ABB RobotStudio station: UiS_E458_nov18_20210914-220803.rsstn

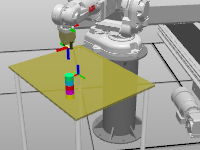
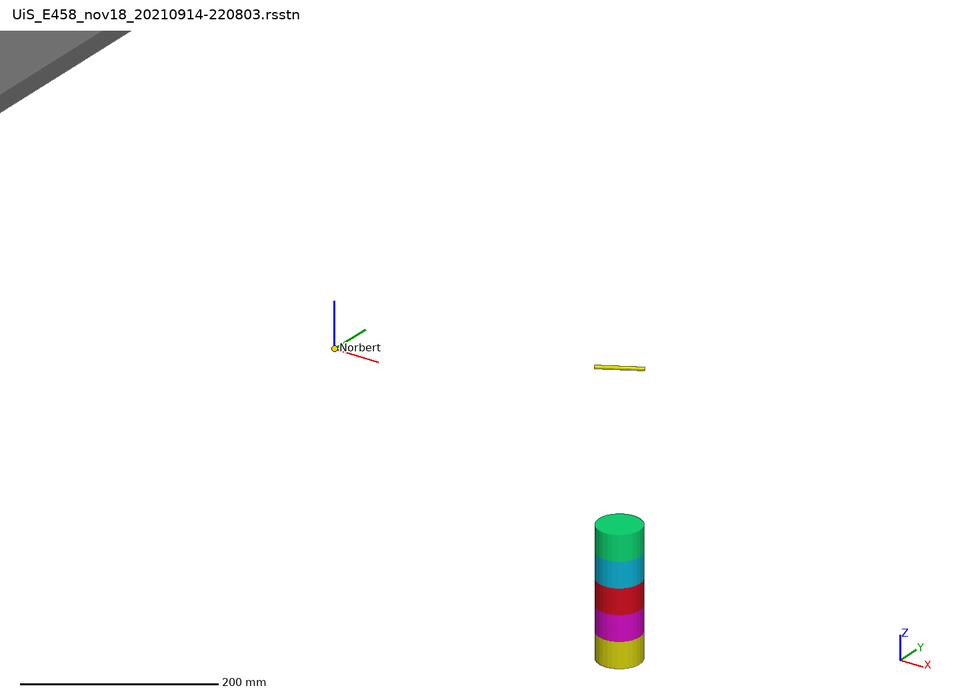
[picture v1: parts stored in the station drawn from their meshes, with robot base, taught points and paths (robot models come from the ABB library and are not in the file)]
Station UiS_E458_nov18 (saved by RobotStudio 21.2.9526.0)
Controller Norbert, task T_ROB1: task frame (RAPID world) sits at (-305, -752, 720) mm, rotated rx 0 ry 0 rz 30 deg in the station
Controller Norbert
  mechanical unit ROB_1: Norbert, 6 joints, base frame (0, 0, 0) mm
Layout (positions relative to the parent item):
  - PedestalN [part, from Libraries\Pedestal.rslib] at (-305, -752, 0) mm, rotated rx 0 ry 0 rz -150 deg
  - Conveyor [part, from Libraries\Conveyor.rslib] at (-998.97, -64.27, 615.81) mm, rotated rx 90 ry 0 rz -90 deg
  - Windowtable [part], size 500 x 2400 x 20 mm
  - TableN [part, from Libraries\Desk.rslib] at (-421.89, -1050.54, 0) mm, rotated rx 0 ry 0 rz -60 deg
  - SC_Gripper [smart component, from Libraries\SC_Gripper.rslib] at (348.11, -1183.22, 1162.25) mm, rotated rx 180 ry 0 rz 120 deg
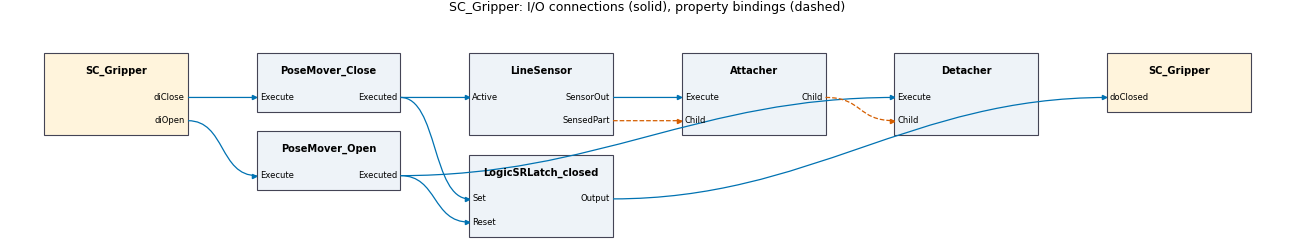
      connections:
        SC_Gripper.diClose -> PoseMover_Close.Execute
        PoseMover_Close.Executed -> LogicSRLatch_closed.Set
        SC_Gripper.diOpen -> PoseMover_Open.Execute
        PoseMover_Open.Executed -> LogicSRLatch_closed.Reset
        LogicSRLatch_closed.Output -> SC_Gripper.doClosed
        PoseMover_Close.Executed -> LineSensor.Active
        LineSensor.SensorOut -> Attacher.Execute
        PoseMover_Open.Executed -> Detacher.Execute
        LineSensor.SensedPart => Attacher.Child
        Attacher.Child => Detacher.Child
    - tGripper [mechanism, from Libraries\SC_Gripper.rslib] at (0, 0, 0) mm; joint values [0.006, 0.006] (rad or m)
    - PoseMover_Close [smart component, from Components\PoseMover.rslib]
        properties: Mechanism=tGripper; Pose=2; Duration=1
    - LogicSRLatch_closed [smart component, from Components\LogicSRLatch.rslib]
    - PoseMover_Open [smart component, from Components\PoseMover.rslib]
        properties: Mechanism=tGripper; Pose=1; Duration=1
    - LineSensor [smart component, from Components\LineSensor.rslib]
        properties: Start=[-5.20417042793042E-18 -0.0255 0.10825]; End=[-2.47198095326695E-17 0.0255 0.10825]; Radius=0.002; SensedPart=Puck1; SensedPoint=[-0.0198517456054688 -1.39565979003906 0.744]
      - _sensorPart_ [part], size 4 x 51 x 4 mm
    - Attacher [smart component, from Components\Attacher.rslib]
        properties: Parent=tGripper; Flange=0; Child=Puck1; Mount=false; Offset=[0 0 0]; Orientation=[0 0 0]
    - Detacher [smart component, from Components\Detacher.rslib]
        properties: Child=Puck1; KeepPosition=true
  - Norbert [mechanism, from Robots\IRB140_6_81_C_G_03.rslib] at (-305, -752, 720) mm, rotated rx 0 ry 0 rz 30 deg; joint values [-1.1071, 1.1816, -1.2308, 0, 1.6199, 0.4636] (rad or m)
  - Puck1 [part] at (348.16, -1183.3, 848) mm, rotated rx 0 ry 0 rz -60 deg, size 50 x 49.9 x 30 mm
  - Puck2 [part] at (348.16, -1183.3, 818) mm, rotated rx 0 ry 0 rz -60 deg, size 50 x 49.9 x 30 mm
  - Puck3 [part] at (348.16, -1183.3, 788) mm, rotated rx 0 ry 0 rz -60 deg, size 50 x 49.9 x 30 mm
  - Puck4 [part] at (348.16, -1183.3, 758) mm, rotated rx 0 ry 0 rz -60 deg, size 50 x 49.9 x 30 mm
  - Puck5 [part] at (348.16, -1183.3, 728) mm, rotated rx 0 ry 0 rz -60 deg, size 50 x 49.9 x 30 mm
Attachment: TableN is attached to PedestalN
Attachment: SC_Gripper is attached to Norbert / Link6
Station signals: DI doClose, DI doOpen
Station logic (signal -> signal, property => property):
  Norbert.doOpen -> SC_Gripper.diOpen
  Norbert.doClose -> SC_Gripper.diClose
  SC_Gripper.doClosed -> Norbert.diClosed
Targets, tools, work objects and paths stored in the station, written as RAPID:
! task T_ROB1
MODULE gripper
  PERS tooldata tGripper:=[TRUE,[[0,0,114.25],[0,0,0,1]],[1,[-0.095984607,0.082520613,38.69176324],[1,0,0,0],0,0,0]];
ENDMODULE

! task T_ROB1
MODULE E458GripperTest
  TASK PERS wobjdata wobjTableN:=[FALSE,TRUE,"",[[150,-500,8],[0.707106781,0,0,-0.707106781]],[[0,0,0],[1,0,0,0]]];
  CONST robtarget target_K0:=[[0,0,0],[0,1,0,0],[-1,0,0,0],[9E+09,9E+09,9E+09,9E+09,9E+09,9E+09]];
  PROC main()
  ENDPROC
  PROC movePuck()
    MoveJ Offs(initialPos, 0, 0, 200),v500,z10,tGripper\WObj:=wobjTableN;
    WaitTime 1.0;
    MoveJ Offs(initialPos, 0, 0, 200),v500,z10,tGripper\WObj:=wobjTableN;
    WaitTime 1.0;
    MoveJ Offs(initialPos, 0, 0, 200),v500,z10,tGripper\WObj:=wobjTableN;
    WaitTime 1.0;
  ENDPROC
ENDMODULE

! task T_ROB1
MODULE LINKEDM
  PROC Linked_m()
  ENDPROC
ENDMODULE

! task T_ROB1
MODULE E458PenTest
  PERS tooldata tSimplePen:=[TRUE,[[0,0,110],[1,0,0,0]],[1,[0,0,1],[1,0,0,0],0,0,0]];
  PROC main()
    Path_10;
  ENDPROC
  PROC Path_10()
  ENDPROC
ENDMODULE

! task T_ROB1
MODULE LINKEDM
  PROC Linked_m()
  ENDPROC
ENDMODULE

